{attribute 'qualified_only'}
{attribute 'strict'}
TYPE E_LampType :
(
	Unknown := -1,
	SetDirect := 0,
	OnOff := 1,
	UpDown := 2
) := Unknown;
END_TYPE

(* stored: Version 1.1.0.1, ProductVersion 3.1.4024.6
   DUT E_LampType: Id {d5912a27-7005-48d6-8ec1-64ec1ff008a0} *)
